TYPE ST_CoeEntry_STRING EXTENDS ST_CoeEntry :
STRUCT
	Value	: Tc2_System.T_MaxString;
END_STRUCT
END_TYPE

(* stored: Version 1.1.0.1, ProductVersion 3.1.4024.13
   DUT ST_CoeEntry_STRING: Id {6a78a22b-6ba5-0e36-37a2-3d07a602e18e} *)
